// TIA Portal V19 export
VAR_GLOBAL   // PLC tag table "02_SAFETY_SINAMICS_A01"
   JBWelderTorch_StsIn AT %I546.0 : "udt_LDrvSafe_typeSinaSTlg30Status";
   JBWelderTorch_CtrlOut AT %Q546.0 : "udt_LDrvSafe_typeSinaSTlg30Control";
   JBPinchRoll_StsIn AT %I552.0 : "udt_LDrvSafe_typeSinaSTlg30Status";
   JBPinchRoll_CtrlOut AT %Q552.0 : "udt_LDrvSafe_typeSinaSTlg30Control";
   Straightener_StsIn AT %I288.0 : "udt_LDrvSafe_typeSinaSTlg30Status";
   Straightener_CtrlOut AT %Q288.0 : "udt_LDrvSafe_typeSinaSTlg30Control";
   DecoilersTranslation_StsIn AT %I526.0 : "udt_LDrvSafe_typeSinaSTlg30Status";
   DecoilersTranslation_CtrlOut AT %Q526.0 : "udt_LDrvSafe_typeSinaSTlg30Control";
   Decoiler1_StsIn AT %I510.0 : "udt_LDrvSafe_typeSinaSTlg30Status";
   Decoiler1_CtrlOut AT %Q510.0 : "udt_LDrvSafe_typeSinaSTlg30Control";
   Decoiler2_StsIn AT %I516.0 : "udt_LDrvSafe_typeSinaSTlg30Status";
   Decoiler2_CtrlOut AT %Q516.0 : "udt_LDrvSafe_typeSinaSTlg30Control";
   CoilCar_StsIn AT %I536.0 : "udt_LDrvSafe_typeSinaSTlg30Status";
   CoilCar_CtrlOut AT %Q536.0 : "udt_LDrvSafe_typeSinaSTlg30Control";
END_VAR
